// Implicitly generated code : DO NOT EDIT
FUNCTION CheckDivLReal : LREAL
VAR_INPUT
    divisor:LREAL;
END_VAR

// Implicitly generated code : Only an Implementation suggestion
{noflow}
IF divisor = 0 THEN
    CheckDivLReal:=1;
ELSE
    CheckDivLReal:=divisor;
END_IF;
{flow}

END_FUNCTION

(* stored: Version 1.1.0.1
   POU CheckDivLReal: Id {a71e081c-e798-4b02-b8e7-849cfc6cac35}, SpecialFunc CheckDivReal64 *)
